PROGRAM Pneumatics_Template
VAR
    //Define all necessary variables for your application
END_VAR
VAR CONSTANT
	cAXIS_ID: USINT := 1;
END_VAR

//Initial parameters of an Pneumatic Axis
//Uncomment the next IF statement to configure and activate the intial parameters of the axis
(*
IF _TaskInfo[fbGetCurTaskIndex.index].FirstCycle THEN
    GVL.astPneumaticAxes[cAXIS_ID].stPneumaticAxisConfig.sPneumaticAxisName := 'P1PneuAxis';
    GVL.astPneumaticAxes[cAXIS_ID].stPneumaticAxisConfig.bSafetyShutter := FALSE;
    GVL.astPneumaticAxes[cAXIS_ID].stPneumaticAxisConfig.nTimeToExtend := 10;
    GVL.astPneumaticAxes[cAXIS_ID].stPneumaticAxisConfig.nTimeToRetract := 10;
    GVL.astPneumaticAxes[cAXIS_ID].stPneumaticAxisConfig.tAllowTimePressureOutOfRange := GVL_APP.tTIME_PRESSURE_OUT_OF_RANGE;
    GVL.astPneumaticAxes[cAXIS_ID].stPneumaticAxisConfig.eSelectPneumaticAxisGroup := E_PneumaticAxisGroup.ePneumaticAxisGroup#;
    GVL.astPneumaticAxes[cAXIS_ID].stPneumaticAxisConfig.fLowLimitPressureValue := GVL_APP.fLOW_LIMIT_AIR_PRESSURE#;
    GVL.astPneumaticAxes[cAXIS_ID].stPneumaticAxisConfig.fHighLimitPressureValue := GVL_APP.fHIGH_LIMIT_AIR_PRESSURE#;
END_IF
*)

END_PROGRAM

(* stored: Version 1.1.0.1
   POU Pneumatics_Template: Id {7bf401fb-a600-4741-a67b-36f20e194cfc}, SpecialFunc None *)
